FUNCTION_BLOCK fbInverterVertHome
VAR_INPUT
	bExecute	: BOOL;
	bEstop		: BOOL;
	bHomeFor	: BOOL;
	bHomeRev	: BOOL;
	bHomeSenser	: BOOL;
	bOTsensor1		: BOOL;
	bOTsensor2		: BOOL;
	bReset			: BOOL;
	i1stRPM			: INT;
	i2ndRPM			: INT;
	rInverterRatio		: REAL;
	EncoderRatio		: LREAL;

END_VAR
VAR_OUTPUT
	bDone		: BOOL;
	bBusy		: BOOL;
	bError		: BOOL;
	bMovForBit	: BOOL;
	bMovRevBit	: BOOL;
	bMovFor2ndBit	: BOOL;
	bMovRev2ndBit	: BOOL;
	bMovFor3rdBit	: BOOL;
	bMovRev3rdBit	: BOOL;
	lrActualPosReference	: LREAL;

END_VAR
VAR_IN_OUT

	iHomeHzout	: INT;
	Axis1		: axis_ref;

END_VAR
VAR
	MCRAP1: MC_ReadActualPosition;
	PowerRelay: TON;
	ArmMovActualPos: LREAL;
	RTRIG1: R_TRIG;
	Move2Home: BOOL;
	HomingStop: BOOL;
	Conv1: AM_InverterConversionHz;
	Conv2: AM_InverterConversionHz;
	CMP1: fbServoPosCmp;
	ArmReachHome: BOOL;
	Conv3: AM_InverterConversionHz;
	Conv4: AM_InverterConversionHz;
	MoveAwayHome: BOOL;
	Conv5: AM_InverterConversionHz;
	Conv6: AM_InverterConversionHz;
	HomingStep1: BOOL;
	MCSPOS1: MC_SetPosition;
	SetPosDone: BOOL;
	TON2: TON;
	T1: TON;
	T2: TON;
	HomeSensorTriggerBit: BOOL;
	HomingStep2: BOOL;
	OTstop: BOOL;
	TRIG1: R_TRIG;
	TRIG2: R_TRIG;
	RTRIG2: R_TRIG;
	i1stRPMTemp: INT;
	i2ndRPMTemp: INT;
	LrPosBeforeConvert: LREAL;
	TON10: TON;
END_VAR

VAR PERSISTENT

	HorzArmPos : LREAL;

END_VAR
VAR // added by the converter: edge detectors and wires of the graphical bodies
    _w1, _w2 : INT;
    _w3 : LREAL;
END_VAR

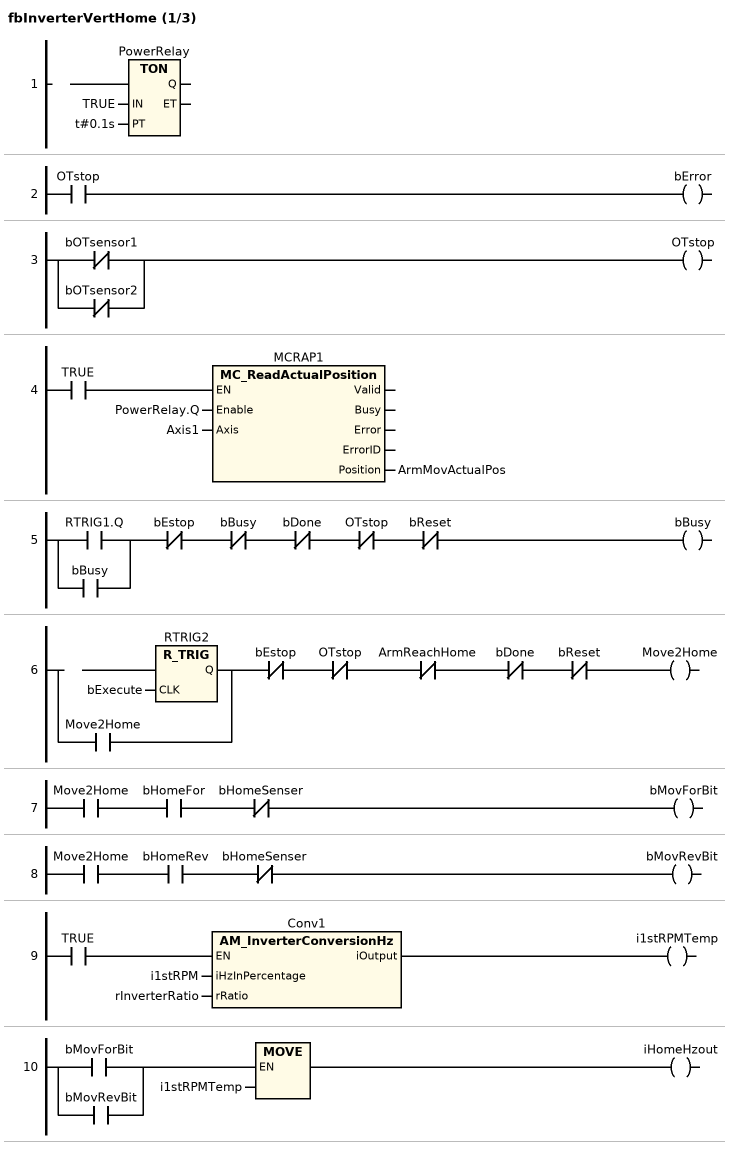
// NETWORK 1
PowerRelay(IN := TRUE, PT := t#0.1s); // TON

// NETWORK 2
bError := OTstop;

// NETWORK 3
OTstop := NOT bOTsensor1 OR NOT bOTsensor2;

// NETWORK 4
MCRAP1(Enable := PowerRelay.Q, Axis := Axis1, Position => ArmMovActualPos); // MC_ReadActualPosition

// NETWORK 5
bBusy := (RTRIG1.Q OR bBusy) AND NOT bEstop AND NOT bBusy AND NOT bDone AND NOT OTstop AND NOT bReset;

// NETWORK 6
RTRIG2(CLK := bExecute); // R_TRIG
Move2Home := (RTRIG2.Q OR Move2Home) AND NOT bEstop AND NOT OTstop AND NOT ArmReachHome AND NOT bDone AND NOT bReset;

// NETWORK 7
bMovForBit := Move2Home AND bHomeFor AND NOT bHomeSenser;

// NETWORK 8
bMovRevBit := Move2Home AND bHomeRev AND NOT bHomeSenser;

// NETWORK 9
Conv1(iHzInPercentage := i1stRPM, rRatio := rInverterRatio); // AM_InverterConversionHz
i1stRPMTemp := Conv1.iOutput;

// NETWORK 10
IF bMovForBit OR bMovRevBit THEN _w1 := i1stRPMTemp; END_IF
iHomeHzout := _w1;

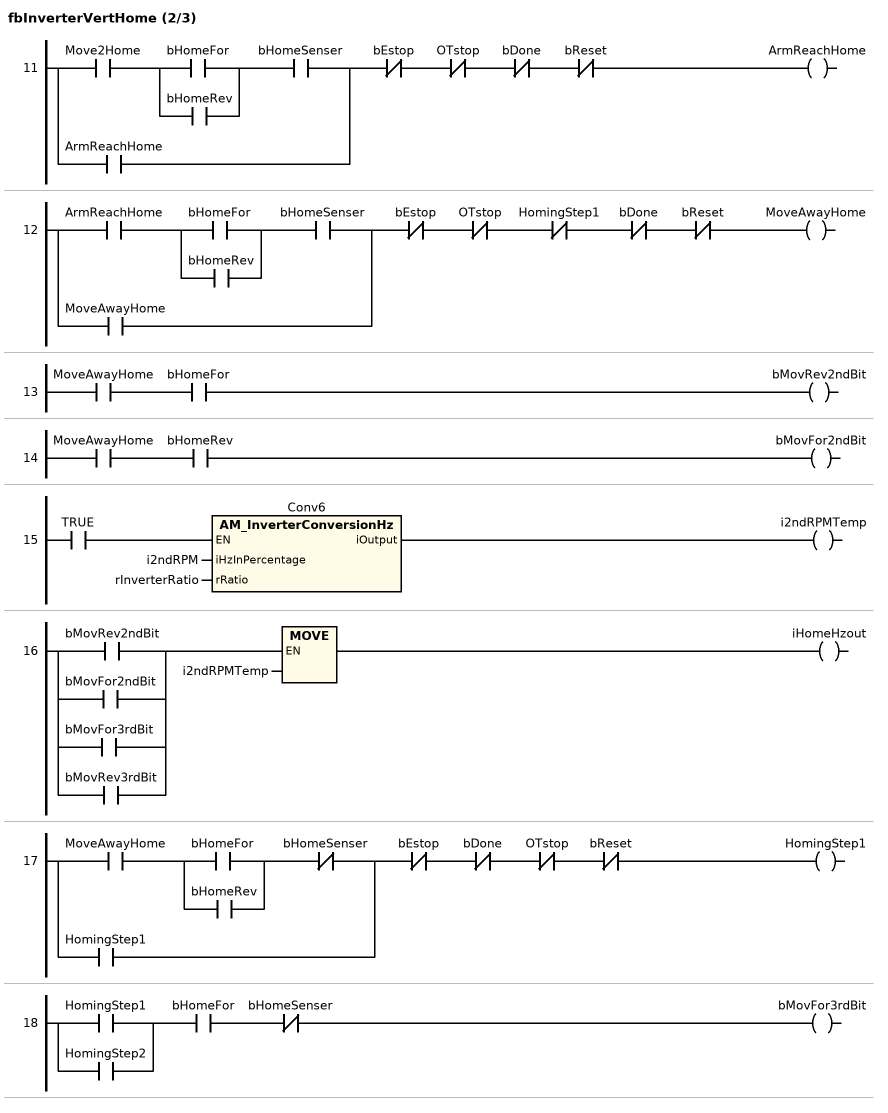
// NETWORK 11
ArmReachHome := ((Move2Home AND (bHomeFor OR bHomeRev)) AND bHomeSenser OR ArmReachHome) AND NOT bEstop AND NOT OTstop AND NOT bDone AND NOT bReset;

// NETWORK 12
MoveAwayHome := ((ArmReachHome AND (bHomeFor OR bHomeRev)) AND bHomeSenser OR MoveAwayHome) AND NOT bEstop AND NOT OTstop AND NOT HomingStep1 AND NOT bDone AND NOT bReset;

// NETWORK 13
bMovRev2ndBit := MoveAwayHome AND bHomeFor;

// NETWORK 14
bMovFor2ndBit := MoveAwayHome AND bHomeRev;

// NETWORK 15
Conv6(iHzInPercentage := i2ndRPM, rRatio := rInverterRatio); // AM_InverterConversionHz
i2ndRPMTemp := Conv6.iOutput;

// NETWORK 16
IF bMovRev2ndBit OR bMovFor2ndBit OR bMovFor3rdBit OR bMovRev3rdBit THEN _w2 := i2ndRPMTemp; END_IF
iHomeHzout := _w2;

// NETWORK 17
HomingStep1 := ((MoveAwayHome AND (bHomeFor OR bHomeRev)) AND NOT bHomeSenser OR HomingStep1) AND NOT bEstop AND NOT bDone AND NOT OTstop AND NOT bReset;

// NETWORK 18
bMovFor3rdBit := (HomingStep1 OR HomingStep2) AND bHomeFor AND NOT bHomeSenser;

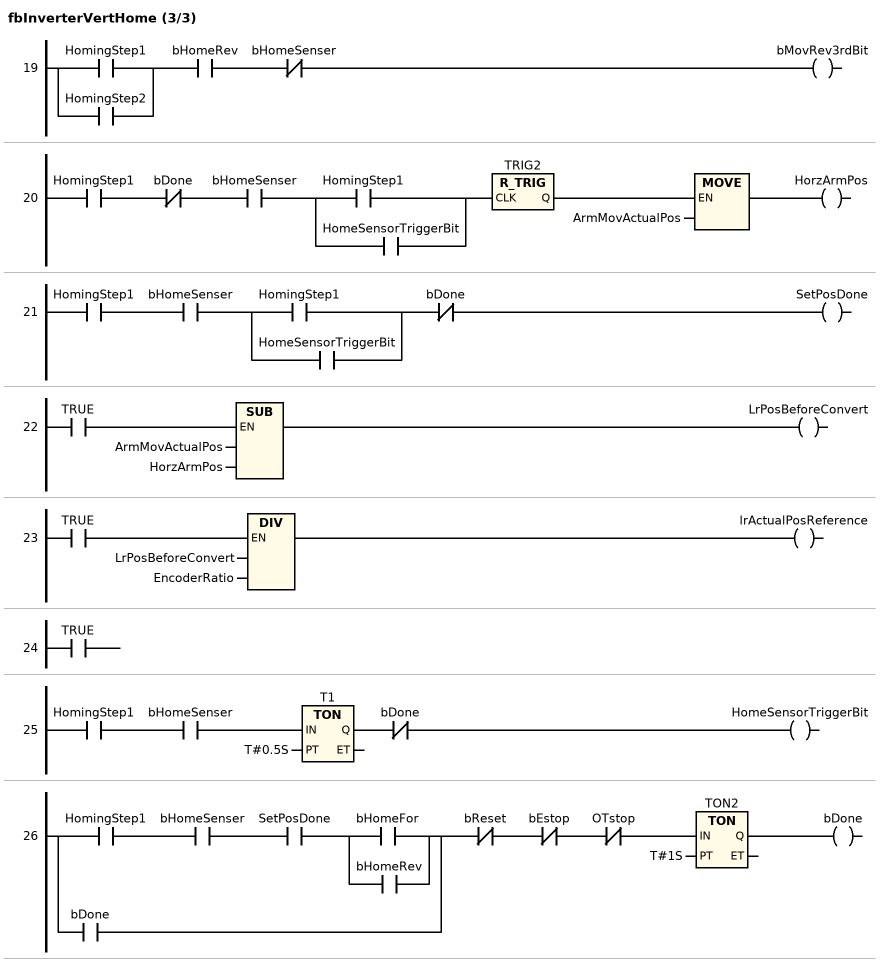
// NETWORK 19
bMovRev3rdBit := (HomingStep1 OR HomingStep2) AND bHomeRev AND NOT bHomeSenser;

// NETWORK 20
TRIG2(CLK := HomingStep1 AND NOT bDone AND bHomeSenser AND (HomingStep1 OR HomeSensorTriggerBit)); // R_TRIG
IF TRIG2.Q THEN _w3 := ArmMovActualPos; END_IF
HorzArmPos := _w3;

// NETWORK 21
SetPosDone := (HomingStep1 AND bHomeSenser AND (HomingStep1 OR HomeSensorTriggerBit)) AND NOT bDone;

// NETWORK 22
LrPosBeforeConvert := ArmMovActualPos - HorzArmPos;

// NETWORK 23
lrActualPosReference := LrPosBeforeConvert / EncoderRatio;

// NETWORK 24

// NETWORK 25
T1(IN := HomingStep1 AND bHomeSenser, PT := T#0.5S); // TON
HomeSensorTriggerBit := T1.Q AND NOT bDone;

// NETWORK 26
TON2(IN := (HomingStep1 AND bHomeSenser AND SetPosDone AND (bHomeFor OR bHomeRev) OR bDone) AND NOT bReset AND NOT bEstop AND NOT OTstop, PT := T#1S); // TON
bDone := TON2.Q;

END_FUNCTION_BLOCK

(* stored: Version 1.1.0.1, ProductVersion 3.1.4024.12
   POU fbInverterVertHome: Id {d3994559-e33c-483e-b385-bc204c2f3d56}, SpecialFunc None *)
